{attribute 'GeneratedUsingTerminal: EKM1101-0000-0016'}
{attribute addProperty BoxType "EKM1101-0000-0016"}
{attribute addProperty Id "DiagBOOL1ErrorBOOL1Input_cycle_CounterBYTE1TxPDO_StateBOOL1IDUSINT1"}
{attribute addProperty CRC "2554836207"}
{attribute addProperty Size "5"}
TYPE Status_9847B4EF :
STRUCT
	{attribute addProperty Name "Diag"}
	Diag : BOOL;
	{attribute addProperty Name "Error"}
	Error : BOOL;
	{attribute addProperty Name "Input_cycle_Counter"}
	Input_cycle_Counter : BYTE;
	{attribute addProperty Name "TxPDO_State"}
	TxPDO_State : BOOL;
	{attribute addProperty Name "ID"}
	ID : USINT;
END_STRUCT
END_TYPE

(* stored: Version 1.2.0.0, ProductVersion 3.1.4024.9
   DUT Status_9847B4EF: Id {f4720c80-19d1-4735-a075-6028160ec062} *)
